// TIA Portal V19 export
FUNCTION "PostPunchingMatCounter_CALL" : Void   // FC159, LAD
// stored: SetENOAutomatically false
BEGIN

REGION Network 1: Coordination IN
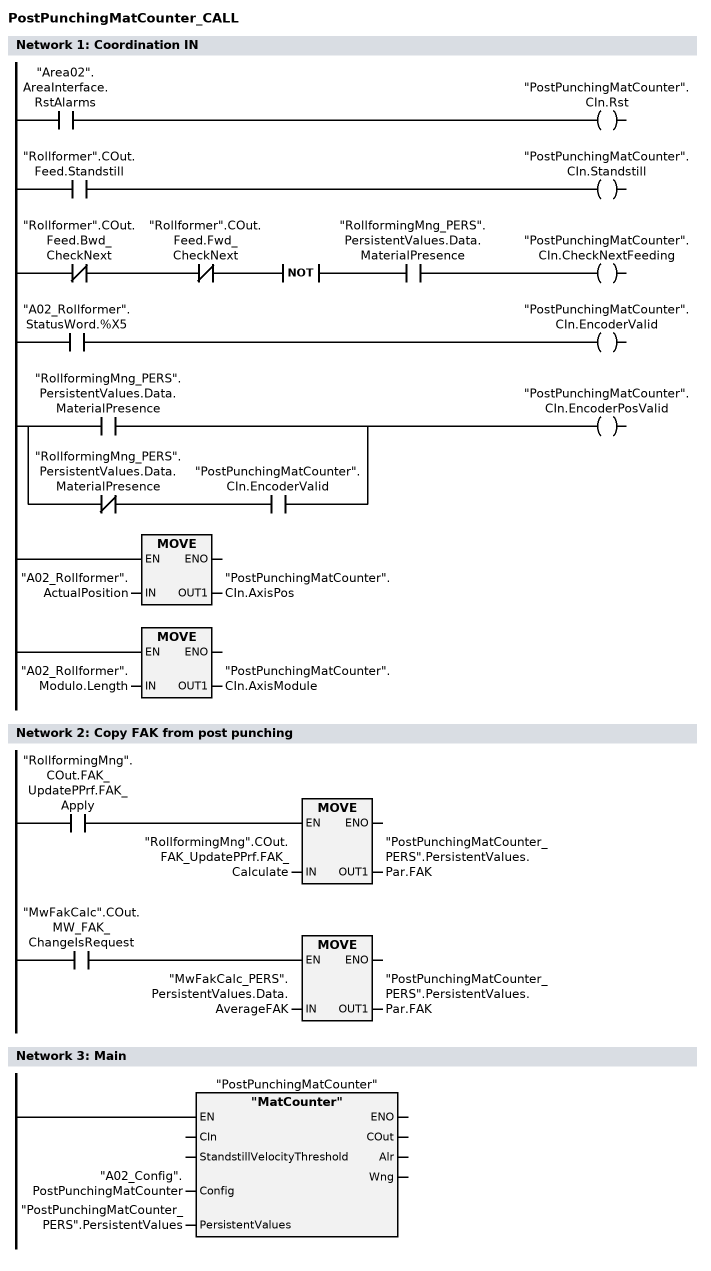
   RUNG wire#powerrail
      Contact( "Area02".AreaInterface.RstAlarms )
      Coil( "PostPunchingMatCounter".CIn.Rst )
   END_RUNG
   RUNG wire#powerrail
      Contact( "Rollformer".COut.Feed.Standstill )
      Coil( "PostPunchingMatCounter".CIn.Standstill )
   END_RUNG
   RUNG wire#powerrail
      I_Contact( "Rollformer".COut.Feed.Bwd_CheckNext )
      I_Contact( "Rollformer".COut.Feed.Fwd_CheckNext )
      Not()
      Contact( "RollformingMng_PERS".PersistentValues.Data.MaterialPresence )
      Coil( "PostPunchingMatCounter".CIn.CheckNextFeeding )
   END_RUNG
   RUNG wire#powerrail
      Contact( "A02_Rollformer".StatusWord.%X5 )
      Coil( "PostPunchingMatCounter".CIn.EncoderValid )
   END_RUNG
   RUNG wire#powerrail
      Contact( "RollformingMng_PERS".PersistentValues.Data.MaterialPresence )
      wire#w1
      Coil( "PostPunchingMatCounter".CIn.EncoderPosValid )
   END_RUNG
   RUNG wire#powerrail
      I_Contact( "RollformingMng_PERS".PersistentValues.Data.MaterialPresence )
      Contact( "PostPunchingMatCounter".CIn.EncoderValid )
   END_RUNG wire#w1
   RUNG wire#powerrail
      Move(in := "A02_Rollformer".ActualPosition, out1 => "PostPunchingMatCounter".CIn.AxisPos)
   END_RUNG
   RUNG wire#powerrail
      Move(in := "A02_Rollformer".Modulo.Length, out1 => "PostPunchingMatCounter".CIn.AxisModule)
   END_RUNG
   // the same network as SCL:
   "PostPunchingMatCounter".CIn.Rst := "Area02".AreaInterface.RstAlarms;
   "PostPunchingMatCounter".CIn.Standstill := "Rollformer".COut.Feed.Standstill;
   "PostPunchingMatCounter".CIn.CheckNextFeeding := NOT (NOT "Rollformer".COut.Feed.Bwd_CheckNext AND NOT "Rollformer".COut.Feed.Fwd_CheckNext) AND "RollformingMng_PERS".PersistentValues.Data.MaterialPresence;
   "PostPunchingMatCounter".CIn.EncoderValid := "A02_Rollformer".StatusWord.%X5;
   "PostPunchingMatCounter".CIn.EncoderPosValid := "RollformingMng_PERS".PersistentValues.Data.MaterialPresence OR (NOT "RollformingMng_PERS".PersistentValues.Data.MaterialPresence AND "PostPunchingMatCounter".CIn.EncoderValid);
   "PostPunchingMatCounter".CIn.AxisPos := "A02_Rollformer".ActualPosition;
   "PostPunchingMatCounter".CIn.AxisModule := "A02_Rollformer".Modulo.Length;
END_REGION

REGION Network 2: Copy FAK from post punching
   RUNG wire#powerrail
      Contact( "RollformingMng".COut.FAK_UpdatePPrf.FAK_Apply )
      Move(in := "RollformingMng".COut.FAK_UpdatePPrf.FAK_Calculate, out1 => "PostPunchingMatCounter_PERS".PersistentValues.Par.FAK)
   END_RUNG
   RUNG wire#powerrail
      Contact( "MwFakCalc".COut.MW_FAK_ChangeIsRequest )
      Move(in := "MwFakCalc_PERS".PersistentValues.Data.AverageFAK, out1 => "PostPunchingMatCounter_PERS".PersistentValues.Par.FAK)
   END_RUNG
   // the same network as SCL:
   IF "RollformingMng".COut.FAK_UpdatePPrf.FAK_Apply THEN
       "PostPunchingMatCounter_PERS".PersistentValues.Par.FAK := "RollformingMng".COut.FAK_UpdatePPrf.FAK_Calculate;
   END_IF;
   IF "MwFakCalc".COut.MW_FAK_ChangeIsRequest THEN
       "PostPunchingMatCounter_PERS".PersistentValues.Par.FAK := "MwFakCalc_PERS".PersistentValues.Data.AverageFAK;
   END_IF;
END_REGION

REGION Network 3: Main
   RUNG wire#powerrail
      "PostPunchingMatCounter"(CIn :=, StandstillVelocityThreshold :=, Config := "A02_Config".PostPunchingMatCounter, PersistentValues := "PostPunchingMatCounter_PERS".PersistentValues, COut =>, Alr =>, Wng =>)
   END_RUNG
   // the same network as SCL:
   "PostPunchingMatCounter"(Config := "A02_Config".PostPunchingMatCounter,   // "MatCounter"
                           PersistentValues := "PostPunchingMatCounter_PERS".PersistentValues);
END_REGION
END_FUNCTION
